PROGRAM MAIN
VAR
	connect: BOOL;
	disconnect: BOOL;
	beep: BOOL;
	queryTargetVoltage: BOOL;
	targetVoltage : LREAL;
END_VAR

serialPort1.CyclicCall();
powerSupply.CyclicCall();

// control of the PSU
IF connect THEN
	connect := FALSE;
	powerSupply.Connect();
END_IF

IF disconnect THEN
	disconnect := FALSE;
	powerSupply.Disconnect();
END_IF

IF beep THEN
	beep := FALSE;
	powerSupply.Beep();
END_IF

IF queryTargetVoltage THEN
	queryTargetVoltage := FALSE;
	powerSupply.QueryTargetVoltage();
END_IF

targetVoltage := powerSupply.TargetVoltage;

END_PROGRAM

(* stored: Version 1.1.0.1, ProductVersion 3.1.4024.9
   POU MAIN: Id {0c120807-b617-41dd-9772-d2e381e423ae}, SpecialFunc None *)
